FUNCTION_BLOCK AX_FB_SR (* Realizes a bistable set-dominat latch (with Adapter) *)
  (* Standard: 61499-1; Description: Copyright (c) 2023 Martin Erich Jobst, HR Agrartechnik GmbH This program and the accompanying materials are made available under the terms of the Eclipse Public License 2.0 which is available at https://www.eclipse.org/legal/epl-2.0/ SPDX-License-Identifier: EPL-2.0 *)
  (* Version 3.0, 2025-04-14, Patrick Aigner, changed package *)
  (* Version 1.0, 2023-04-28, Martin Jobst, initial API and implementation and/or initial documentation *)
  PACKAGE adapter::iec61131::bistableElements;
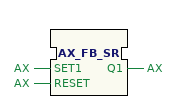
  SOCKETS
    SET1 : adapter::types::unidirectional::AX; (* Set *)
    RESET : adapter::types::unidirectional::AX; (* Reset *)
  END_SOCKETS
  PLUGS
    Q1 : adapter::types::unidirectional::AX; (* Output *)
  END_PLUGS
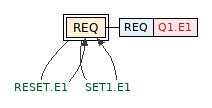
  EC_STATES
    REQ : REQ -> Q1.E1;
  END_STATES
  EC_TRANSITIONS
    REQ TO REQ := SET1.E1;
    REQ TO REQ := RESET.E1;
  END_TRANSITIONS
  ALGORITHM REQ IN ST:
Q1.D1 := SET1.D1 OR ((NOT RESET.D1) AND Q1.D1);
  END_ALGORITHM
END_FUNCTION_BLOCK
